(* Logix 5000 project; controller PLC vendor 1 type 14 code 155 rev 30.14; software revision 30.01; part 2 of 4 *)
(* tags used below, declared in another part *)
   Alarm_Word_Compare : DINT[3];
   Alarm_Word_Current : DINT[3];
   Alarm_Word_New : DINT[3];
   Alarm_Word_Previous : DINT[3];
   Bridge_Timer_Gearing_Duration : TIMER;
   Denester : Denester_R2b;
   Depositor : Depositor_R2b;
   IO : IO_R2a;
   MV_Rate : DINT;
   NC_NF : NCNF_R2a;   // NC/NF BITSHIFTS
   OS : INT[10];
   Rates : Rates_R2b;
   Recipe : Recipe_R2c;
   Recipe_Setpoints_DINT : DINT[23,20];
   Recipe_Setpoints_DINT_Temp : DINT[20];
   Recipe_Setpoints_REAL : REAL[23,20];
   Recipe_Setpoints_REAL_Temp : REAL[20];
   Sequencer_Auto : Sequencer_R2a;
   Sequencer_Home : Sequencer_R2a;
   Servo_MC_Bridge_Shift : Axis_MC_R3b;
   System : System_R2e;
(* MainProgram, continued *)

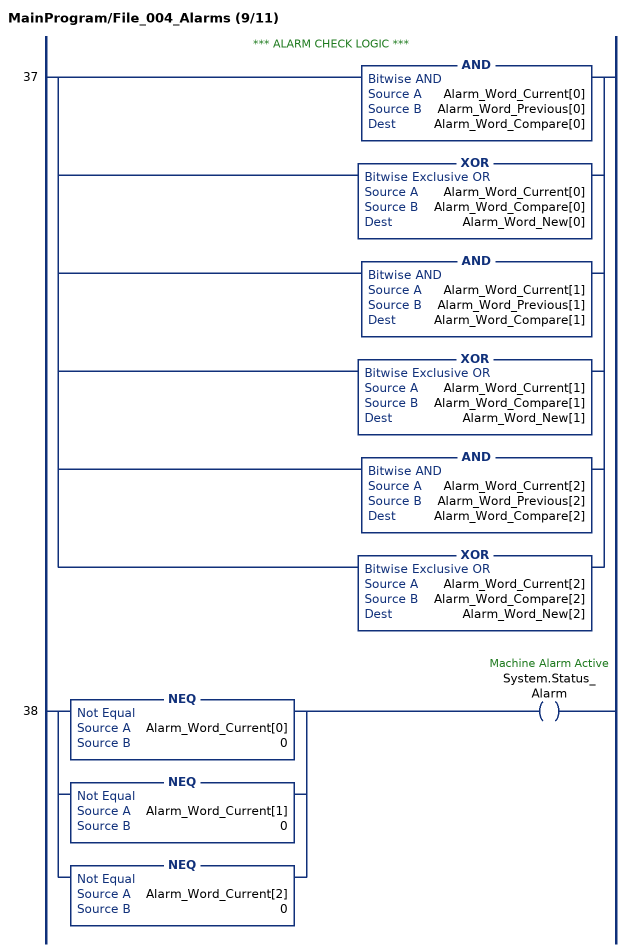
   [picture p24: MainProgram/File_004_Alarms rungs 37-38]
   // *** ALARM CHECK LOGIC ***
   37: [[AND(Alarm_Word_Current[0],Alarm_Word_Previous[0],Alarm_Word_Compare[0]) ,XOR(Alarm_Word_Current[0],Alarm_Word_Compare[0],Alarm_Word_New[0]) ] ,[AND(Alarm_Word_Current[1],Alarm_Word_Previous[1],Alarm_Word_Compare[1]) ,XOR(Alarm_Word_Current[1],Alarm_Word_Compare[1],Alarm_Word_New[1]) ] ,[AND(Alarm_Word_Current[2],Alarm_Word_Previous[2],Alarm_Word_Compare[2]) ,XOR(Alarm_Word_Current[2],Alarm_Word_Compare[2],Alarm_Word_New[2]) ] ];
   38: [NEQ(Alarm_Word_Current[0],0) ,NEQ(Alarm_Word_Current[1],0) ,NEQ(Alarm_Word_Current[2],0) ]OTE(System.Status_Alarm);
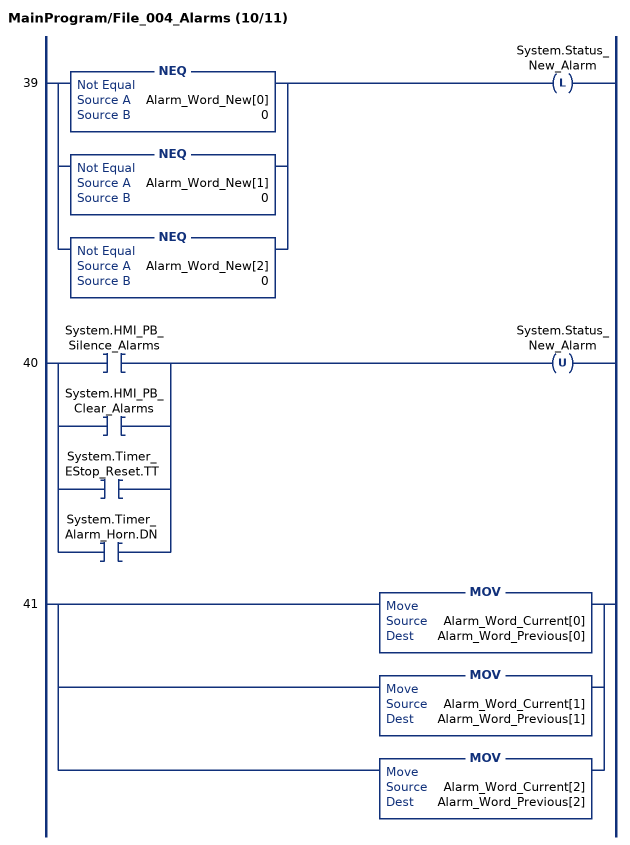
   39: [NEQ(Alarm_Word_New[0],0) ,NEQ(Alarm_Word_New[1],0) ,NEQ(Alarm_Word_New[2],0) ]OTL(System.Status_New_Alarm);
   40: [XIC(System.HMI_PB_Silence_Alarms) ,XIC(System.HMI_PB_Clear_Alarms) ,XIC(System.Timer_EStop_Reset.TT) ,XIC(System.Timer_Alarm_Horn.DN) ]OTU(System.Status_New_Alarm);
   41: [MOV(Alarm_Word_Current[0],Alarm_Word_Previous[0]) ,MOV(Alarm_Word_Current[1],Alarm_Word_Previous[1]) ,MOV(Alarm_Word_Current[2],Alarm_Word_Previous[2]) ];
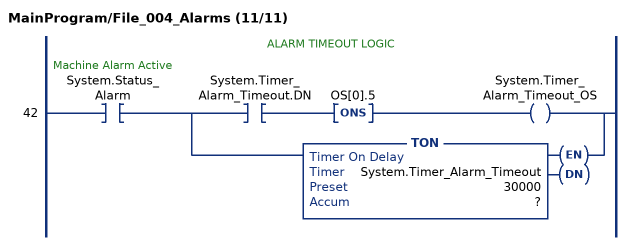
   // ALARM TIMEOUT LOGIC
   42: XIC(System.Status_Alarm)[XIC(System.Timer_Alarm_Timeout.DN) ONS(OS[0].5) OTE(System.Timer_Alarm_Timeout_OS) ,TON(System.Timer_Alarm_Timeout,?,?) ];
END_ROUTINE

ROUTINE File_005_Recipes   (* ladder *)
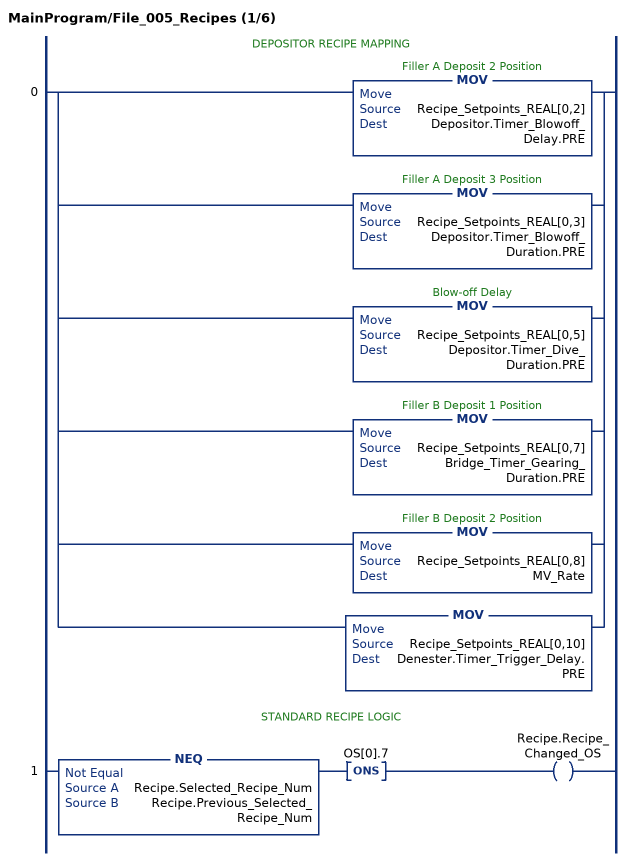
   // DEPOSITOR RECIPE MAPPING
   0: [MOV(Recipe_Setpoints_REAL[0,2],Depositor.Timer_Blowoff_Delay.PRE) ,MOV(Recipe_Setpoints_REAL[0,3],Depositor.Timer_Blowoff_Duration.PRE) ,MOV(Recipe_Setpoints_REAL[0,5],Depositor.Timer_Dive_Duration.PRE) ,MOV(Recipe_Setpoints_REAL[0,7],Bridge_Timer_Gearing_Duration.PRE) ,MOV(Recipe_Setpoints_REAL[0,8],MV_Rate) ,MOV(Recipe_Setpoints_REAL[0,10],Denester.Timer_Trigger_Delay.PRE) ];
   // STANDARD RECIPE LOGIC
   1: NEQ(Recipe.Selected_Recipe_Num,Recipe.Previous_Selected_Recipe_Num)ONS(OS[0].7)OTE(Recipe.Recipe_Changed_OS);
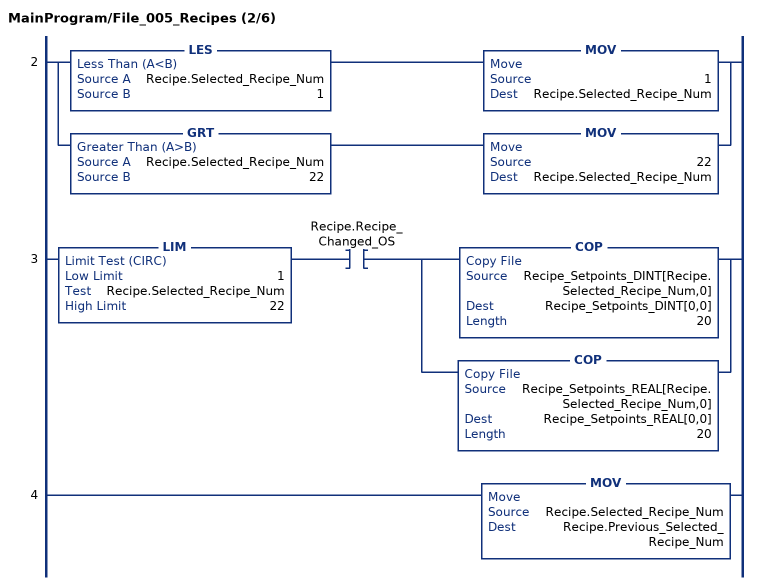
   2: [LES(Recipe.Selected_Recipe_Num,1) MOV(1,Recipe.Selected_Recipe_Num) ,GRT(Recipe.Selected_Recipe_Num,22) MOV(22,Recipe.Selected_Recipe_Num) ];
   3: LIM(1,Recipe.Selected_Recipe_Num,22)XIC(Recipe.Recipe_Changed_OS)[COP(Recipe_Setpoints_DINT[Recipe.Selected_Recipe_Num,0],Recipe_Setpoints_DINT[0,0],20) ,COP(Recipe_Setpoints_REAL[Recipe.Selected_Recipe_Num,0],Recipe_Setpoints_REAL[0,0],20) ];
   4: MOV(Recipe.Selected_Recipe_Num,Recipe.Previous_Selected_Recipe_Num);
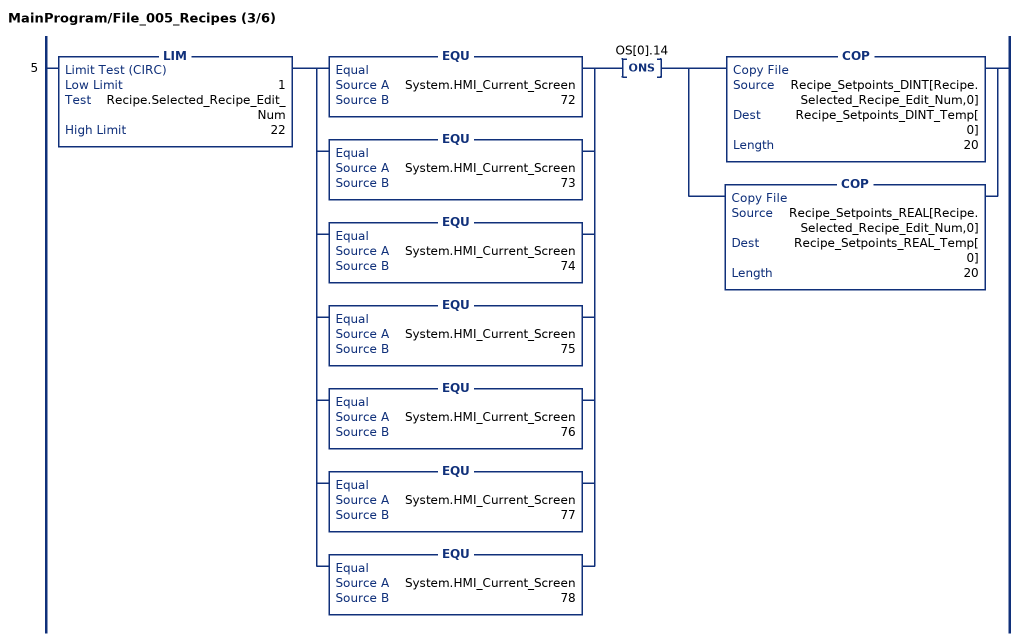
   5: LIM(1,Recipe.Selected_Recipe_Edit_Num,22)[EQU(System.HMI_Current_Screen,72) ,EQU(System.HMI_Current_Screen,73) ,EQU(System.HMI_Current_Screen,74) ,EQU(System.HMI_Current_Screen,75) ,EQU(System.HMI_Current_Screen,76) ,EQU(System.HMI_Current_Screen,77) ,EQU(System.HMI_Current_Screen,78) ]ONS(OS[0].14)[COP(Recipe_Setpoints_DINT[Recipe.Selected_Recipe_Edit_Num,0],Recipe_Setpoints_DINT_Temp[0],20) ,COP(Recipe_Setpoints_REAL[Recipe.Selected_Recipe_Edit_Num,0],Recipe_Setpoints_REAL_Temp[0],20) ];
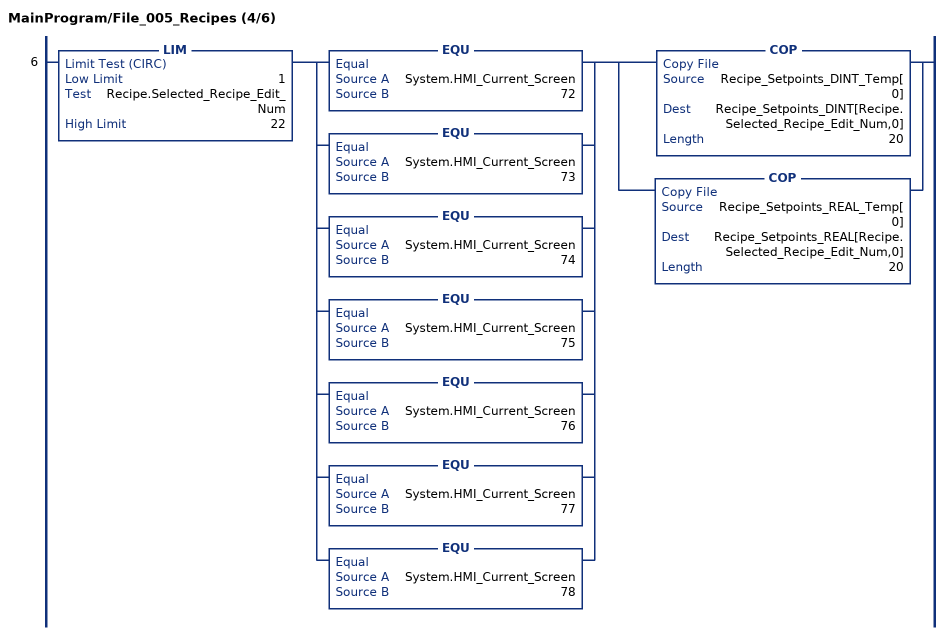
   6: LIM(1,Recipe.Selected_Recipe_Edit_Num,22)[EQU(System.HMI_Current_Screen,72) ,EQU(System.HMI_Current_Screen,73) ,EQU(System.HMI_Current_Screen,74) ,EQU(System.HMI_Current_Screen,75) ,EQU(System.HMI_Current_Screen,76) ,EQU(System.HMI_Current_Screen,77) ,EQU(System.HMI_Current_Screen,78) ][COP(Recipe_Setpoints_DINT_Temp[0],Recipe_Setpoints_DINT[Recipe.Selected_Recipe_Edit_Num,0],20) ,COP(Recipe_Setpoints_REAL_Temp[0],Recipe_Setpoints_REAL[Recipe.Selected_Recipe_Edit_Num,0],20) ];
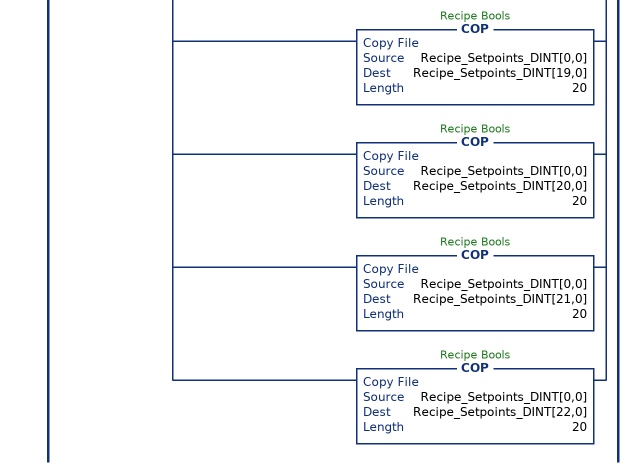
   // RECIPE INITIALIZATION LOGIC
   7: XIC(System.HMI_PB_Recipe_Initialize)[COP(Recipe_Setpoints_DINT[0,0],Recipe_Setpoints_DINT[1,0],20) ,COP(Recipe_Setpoints_DINT[0,0],Recipe_Setpoints_DINT[2,0],20) ,COP(Recipe_Setpoints_DINT[0,0],Recipe_Setpoints_DINT[3,0],20) ,COP(Recipe_Setpoints_DINT[0,0],Recipe_Setpoints_DINT[4,0],20) ,COP(Recipe_Setpoints_DINT[0,0],Recipe_Setpoints_DINT[5,0],20) ,COP(Recipe_Setpoints_DINT[0,0],Recipe_Setpoints_DINT[6,0],20) ,COP(Recipe_Setpoints_DINT[0,0],Recipe_Setpoints_DINT[7,0],20) ,COP(Recipe_Setpoints_DINT[0,0],Recipe_Setpoints_DINT[8,0],20) ,COP(Recipe_Setpoints_DINT[0,0],Recipe_Setpoints_DINT[9,0],20) ,COP(Recipe_Setpoints_DINT[0,0],Recipe_Setpoints_DINT[10,0],20) ,COP(Recipe_Setpoints_DINT[0,0],Recipe_Setpoints_DINT[11,0],20) ,COP(Recipe_Setpoints_DINT[0,0],Recipe_Setpoints_DINT[12,0],20) ,COP(Recipe_Setpoints_DINT[0,0],Recipe_Setpoints_DINT[13,0],20) ,COP(Recipe_Setpoints_DINT[0,0],Recipe_Setpoints_DINT[14,0],20) ,COP(Recipe_Setpoints_DINT[0,0],Recipe_Setpoints_DINT[15,0],20) ,COP(Recipe_Setpoints_DINT[0,0],Recipe_Setpoints_DINT[16,0],20) ,COP(Recipe_Setpoints_DINT[0,0],Recipe_Setpoints_DINT[17,0],20) ,COP(Recipe_Setpoints_DINT[0,0],Recipe_Setpoints_DINT[18,0],20) ,COP(Recipe_Setpoints_DINT[0,0],Recipe_Setpoints_DINT[19,0],20) ,COP(Recipe_Setpoints_DINT[0,0],Recipe_Setpoints_DINT[20,0],20) ,COP(Recipe_Setpoints_DINT[0,0],Recipe_Setpoints_DINT[21,0],20) ,COP(Recipe_Setpoints_DINT[0,0],Recipe_Setpoints_DINT[22,0],20) ];
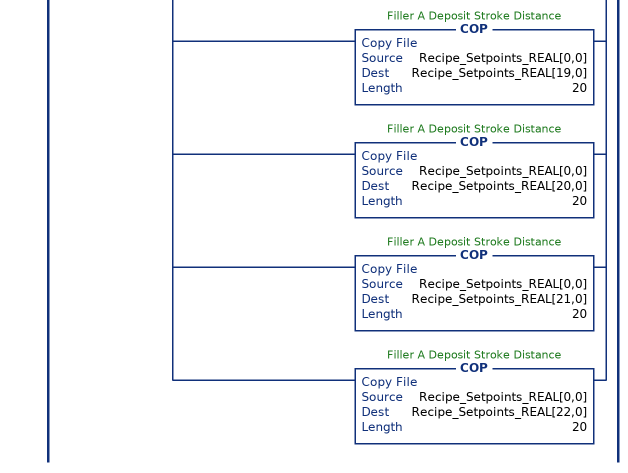
   8: XIC(System.HMI_PB_Recipe_Initialize)[COP(Recipe_Setpoints_REAL[0,0],Recipe_Setpoints_REAL[1,0],20) ,COP(Recipe_Setpoints_REAL[0,0],Recipe_Setpoints_REAL[2,0],20) ,COP(Recipe_Setpoints_REAL[0,0],Recipe_Setpoints_REAL[3,0],20) ,COP(Recipe_Setpoints_REAL[0,0],Recipe_Setpoints_REAL[4,0],20) ,COP(Recipe_Setpoints_REAL[0,0],Recipe_Setpoints_REAL[5,0],20) ,COP(Recipe_Setpoints_REAL[0,0],Recipe_Setpoints_REAL[6,0],20) ,COP(Recipe_Setpoints_REAL[0,0],Recipe_Setpoints_REAL[7,0],20) ,COP(Recipe_Setpoints_REAL[0,0],Recipe_Setpoints_REAL[8,0],20) ,COP(Recipe_Setpoints_REAL[0,0],Recipe_Setpoints_REAL[9,0],20) ,COP(Recipe_Setpoints_REAL[0,0],Recipe_Setpoints_REAL[10,0],20) ,COP(Recipe_Setpoints_REAL[0,0],Recipe_Setpoints_REAL[11,0],20) ,COP(Recipe_Setpoints_REAL[0,0],Recipe_Setpoints_REAL[12,0],20) ,COP(Recipe_Setpoints_REAL[0,0],Recipe_Setpoints_REAL[13,0],20) ,COP(Recipe_Setpoints_REAL[0,0],Recipe_Setpoints_REAL[14,0],20) ,COP(Recipe_Setpoints_REAL[0,0],Recipe_Setpoints_REAL[15,0],20) ,COP(Recipe_Setpoints_REAL[0,0],Recipe_Setpoints_REAL[16,0],20) ,COP(Recipe_Setpoints_REAL[0,0],Recipe_Setpoints_REAL[17,0],20) ,COP(Recipe_Setpoints_REAL[0,0],Recipe_Setpoints_REAL[18,0],20) ,COP(Recipe_Setpoints_REAL[0,0],Recipe_Setpoints_REAL[19,0],20) ,COP(Recipe_Setpoints_REAL[0,0],Recipe_Setpoints_REAL[20,0],20) ,COP(Recipe_Setpoints_REAL[0,0],Recipe_Setpoints_REAL[21,0],20) ,COP(Recipe_Setpoints_REAL[0,0],Recipe_Setpoints_REAL[22,0],20) ];
END_ROUTINE

ROUTINE File_006_Status   (* ladder *)
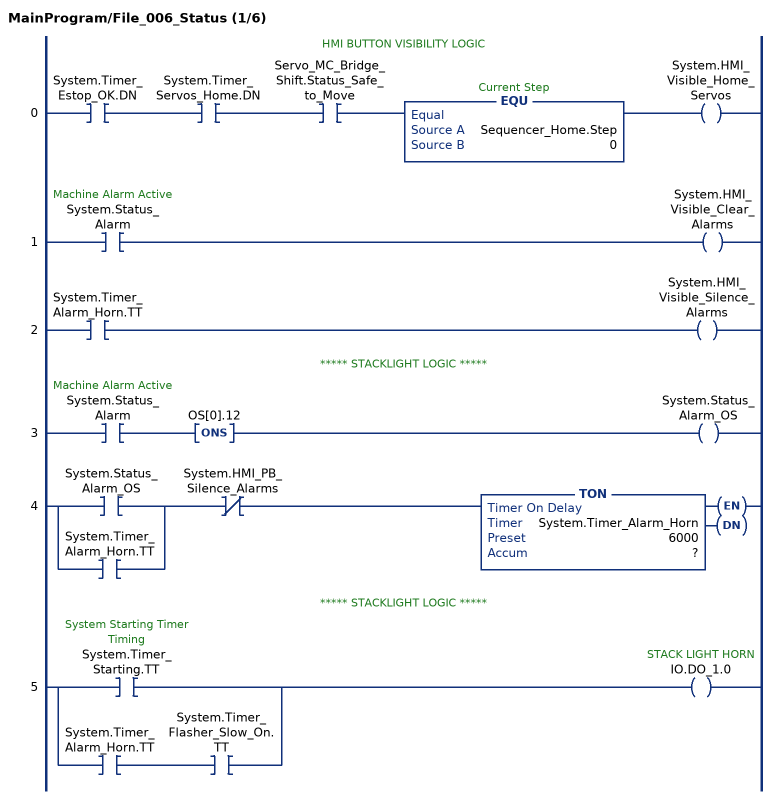
   // HMI BUTTON VISIBILITY LOGIC
   0: XIC(System.Timer_Estop_OK.DN)XIC(System.Timer_Servos_Home.DN)XIC(Servo_MC_Bridge_Shift.Status_Safe_to_Move)EQU(Sequencer_Home.Step,0)OTE(System.HMI_Visible_Home_Servos);
   1: XIC(System.Status_Alarm)OTE(System.HMI_Visible_Clear_Alarms);
   2: XIC(System.Timer_Alarm_Horn.TT)OTE(System.HMI_Visible_Silence_Alarms);
   // ***** STACKLIGHT LOGIC *****
   3: XIC(System.Status_Alarm)ONS(OS[0].12)OTE(System.Status_Alarm_OS);
   4: [XIC(System.Status_Alarm_OS) ,XIC(System.Timer_Alarm_Horn.TT) ]XIO(System.HMI_PB_Silence_Alarms)TON(System.Timer_Alarm_Horn,?,?);
   // ***** STACKLIGHT LOGIC *****
   5: [XIC(System.Timer_Starting.TT) ,XIC(System.Timer_Alarm_Horn.TT) XIC(System.Timer_Flasher_Slow_On.TT) ]OTE(IO.DO_1.0);
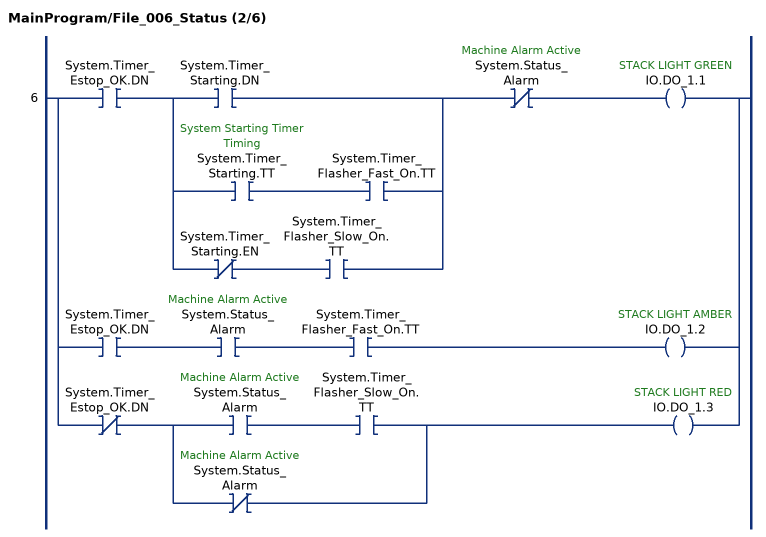
   6: [XIC(System.Timer_Estop_OK.DN) [XIC(System.Timer_Starting.DN) ,XIC(System.Timer_Starting.TT) XIC(System.Timer_Flasher_Fast_On.TT) ,XIO(System.Timer_Starting.EN) XIC(System.Timer_Flasher_Slow_On.TT) ] XIO(System.Status_Alarm) OTE(IO.DO_1.1) ,XIC(System.Timer_Estop_OK.DN) XIC(System.Status_Alarm) XIC(System.Timer_Flasher_Fast_On.TT) OTE(IO.DO_1.2) ,XIO(System.Timer_Estop_OK.DN) [XIC(System.Status_Alarm) XIC(System.Timer_Flasher_Slow_On.TT) ,XIO(System.Status_Alarm) ] OTE(IO.DO_1.3) ];
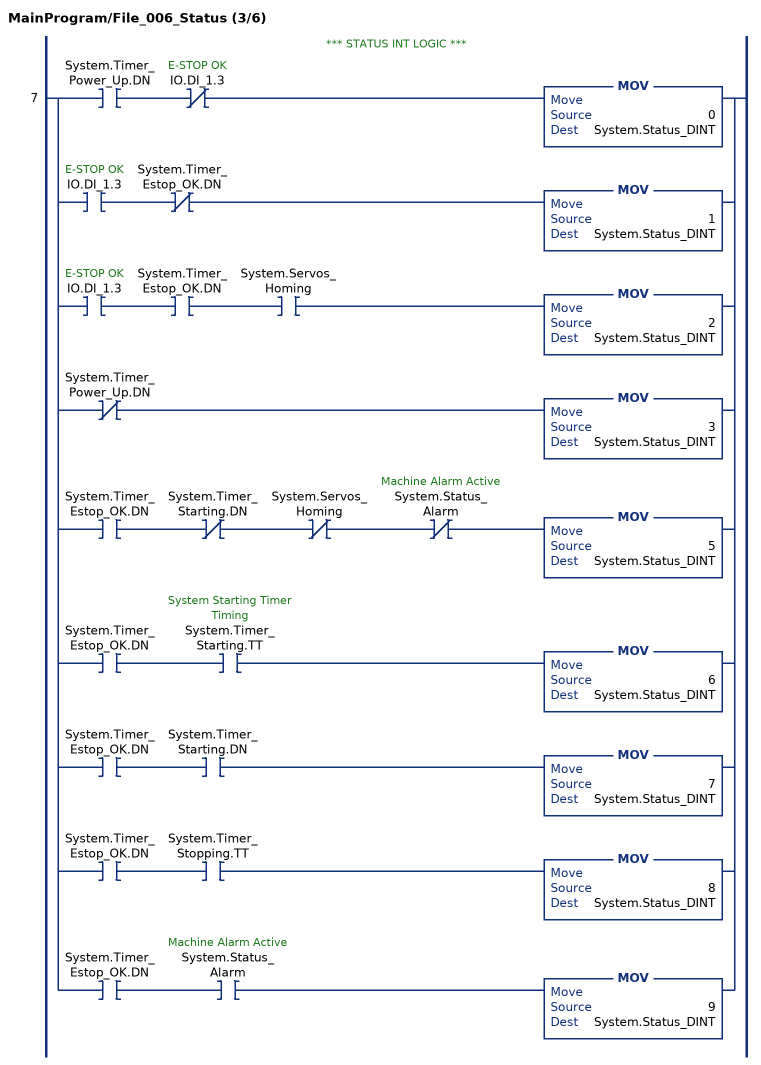
   // *** STATUS INT LOGIC ***
   7: [XIC(System.Timer_Power_Up.DN) XIO(IO.DI_1.3) MOV(0,System.Status_DINT) ,XIC(IO.DI_1.3) XIO(System.Timer_Estop_OK.DN) MOV(1,System.Status_DINT) ,XIC(IO.DI_1.3) XIC(System.Timer_Estop_OK.DN) XIC(System.Servos_Homing) MOV(2,System.Status_DINT) ,XIO(System.Timer_Power_Up.DN) MOV(3,System.Status_DINT) ,XIC(System.Timer_Estop_OK.DN) XIO(System.Timer_Starting.DN) XIO(System.Servos_Homing) XIO(System.Status_Alarm) MOV(5,System.Status_DINT) ,XIC(System.Timer_Estop_OK.DN) XIC(System.Timer_Starting.TT) MOV(6,System.Status_DINT) ,XIC(System.Timer_Estop_OK.DN) XIC(System.Timer_Starting.DN) MOV(7,System.Status_DINT) ,XIC(System.Timer_Estop_OK.DN) XIC(System.Timer_Stopping.TT) MOV(8,System.Status_DINT) ,XIC(System.Timer_Estop_OK.DN) XIC(System.Status_Alarm) MOV(9,System.Status_DINT) ];
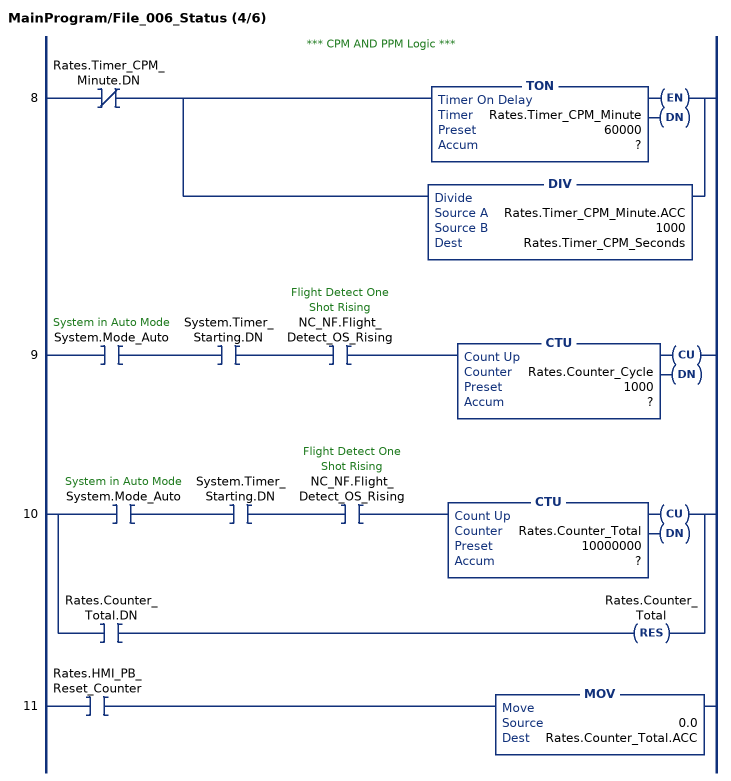
   // *** CPM AND PPM Logic ***
   8: XIO(Rates.Timer_CPM_Minute.DN)[TON(Rates.Timer_CPM_Minute,?,?) ,DIV(Rates.Timer_CPM_Minute.ACC,1000,Rates.Timer_CPM_Seconds) ];
   9: XIC(System.Mode_Auto)XIC(System.Timer_Starting.DN)XIC(NC_NF.Flight_Detect_OS_Rising)CTU(Rates.Counter_Cycle,?,?);
   10: [XIC(System.Mode_Auto) XIC(System.Timer_Starting.DN) XIC(NC_NF.Flight_Detect_OS_Rising) CTU(Rates.Counter_Total,?,?) ,XIC(Rates.Counter_Total.DN) RES(Rates.Counter_Total) ];
   11: XIC(Rates.HMI_PB_Reset_Counter)MOV(0.0,Rates.Counter_Total.ACC);
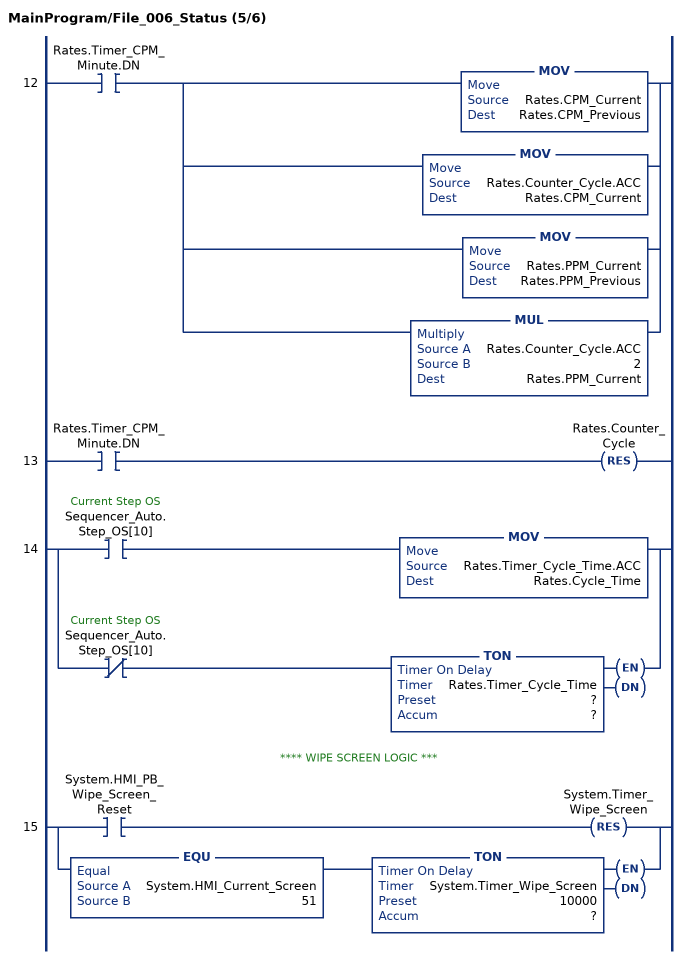
   12: XIC(Rates.Timer_CPM_Minute.DN)[MOV(Rates.CPM_Current,Rates.CPM_Previous) ,MOV(Rates.Counter_Cycle.ACC,Rates.CPM_Current) ,MOV(Rates.PPM_Current,Rates.PPM_Previous) ,MUL(Rates.Counter_Cycle.ACC,2,Rates.PPM_Current) ];
   13: XIC(Rates.Timer_CPM_Minute.DN)RES(Rates.Counter_Cycle);
   14: [XIC(Sequencer_Auto.Step_OS[10]) MOV(Rates.Timer_Cycle_Time.ACC,Rates.Cycle_Time) ,XIO(Sequencer_Auto.Step_OS[10]) TON(Rates.Timer_Cycle_Time,?,?) ];
   // **** WIPE SCREEN LOGIC ***
   15: [XIC(System.HMI_PB_Wipe_Screen_Reset) RES(System.Timer_Wipe_Screen) ,EQU(System.HMI_Current_Screen,51) TON(System.Timer_Wipe_Screen,?,?) ];
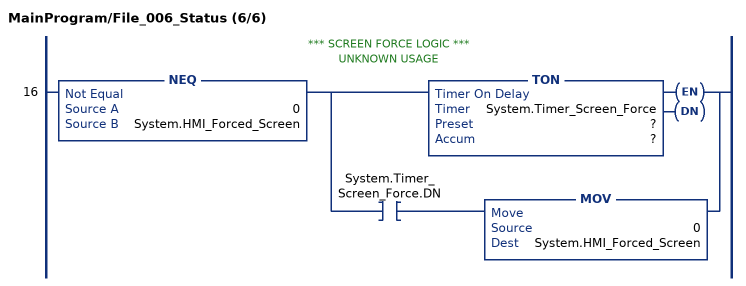
   // *** SCREEN FORCE LOGIC ***
   // UNKNOWN USAGE
   16: NEQ(0,System.HMI_Forced_Screen)[TON(System.Timer_Screen_Force,?,?) ,XIC(System.Timer_Screen_Force.DN) MOV(0,System.HMI_Forced_Screen) ];
END_ROUTINE

ROUTINE File_007_NC_NF   (* ladder *)
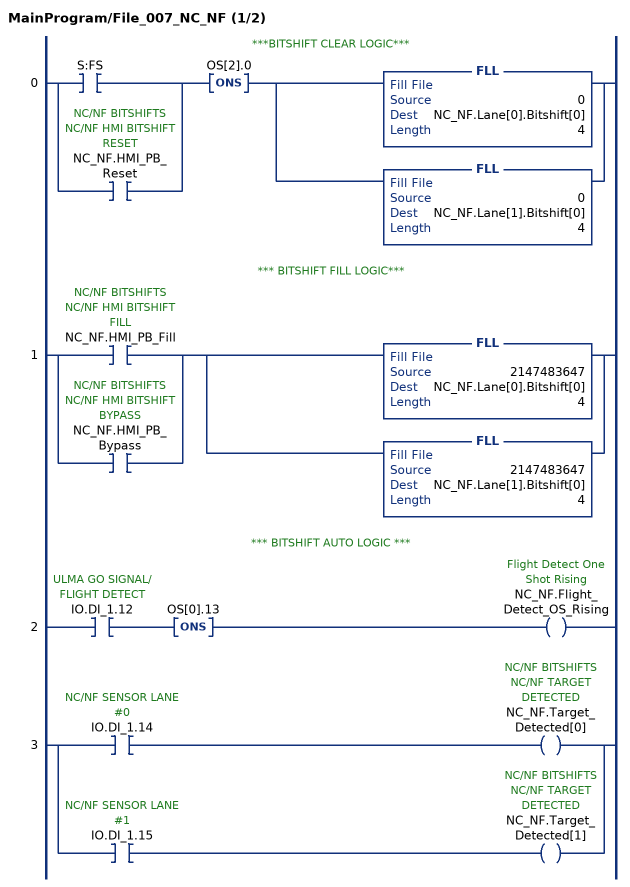
   // ***BITSHIFT CLEAR LOGIC***
   0: [XIC(S:FS) ,XIC(NC_NF.HMI_PB_Reset) ]ONS(OS[2].0)[FLL(0,NC_NF.Lane[0].Bitshift[0],4) ,FLL(0,NC_NF.Lane[1].Bitshift[0],4) ];
   // *** BITSHIFT FILL LOGIC***
   1: [XIC(NC_NF.HMI_PB_Fill) ,XIC(NC_NF.HMI_PB_Bypass) ][FLL(2147483647,NC_NF.Lane[0].Bitshift[0],4) ,FLL(2147483647,NC_NF.Lane[1].Bitshift[0],4) ];
   // *** BITSHIFT AUTO LOGIC ***
   2: XIC(IO.DI_1.12)ONS(OS[0].13)OTE(NC_NF.Flight_Detect_OS_Rising);
   3: [XIC(IO.DI_1.14) OTE(NC_NF.Target_Detected[0]) ,XIC(IO.DI_1.15) OTE(NC_NF.Target_Detected[1]) ];
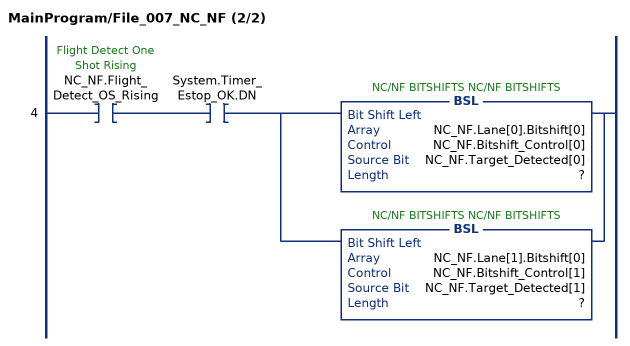
   4: XIC(NC_NF.Flight_Detect_OS_Rising)XIC(System.Timer_Estop_OK.DN)[BSL(NC_NF.Lane[0].Bitshift[0],NC_NF.Bitshift_Control[0],NC_NF.Target_Detected[0],?) ,BSL(NC_NF.Lane[1].Bitshift[0],NC_NF.Bitshift_Control[1],NC_NF.Target_Detected[1],?) ];
END_ROUTINE

ROUTINE File_010_Digital_Inputs   (* ladder *)
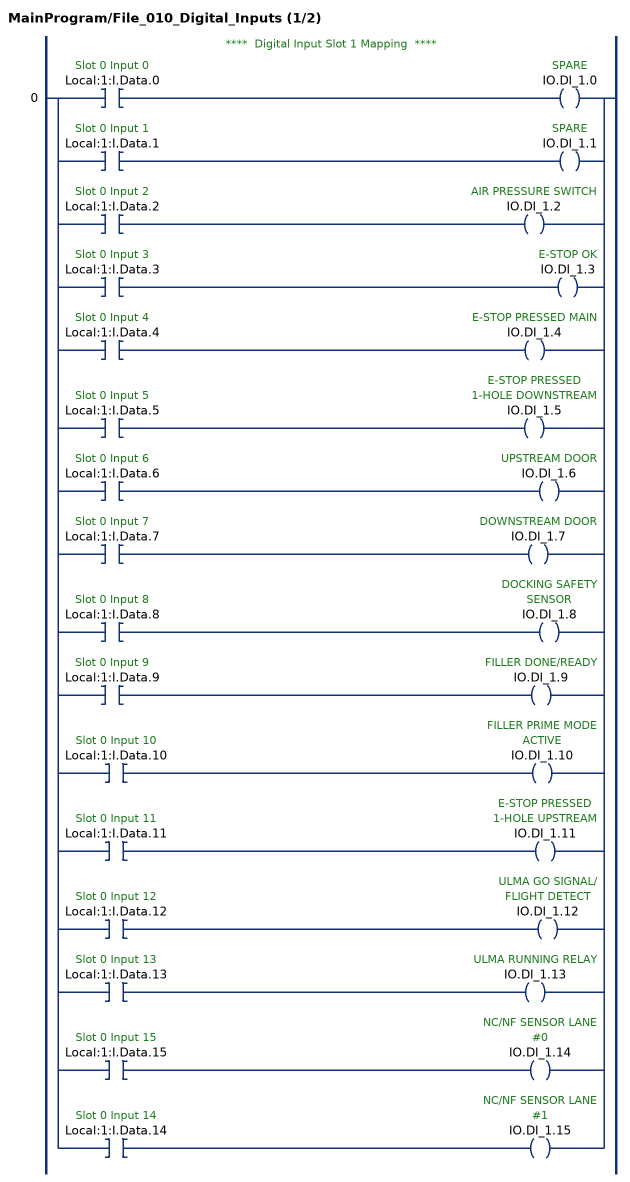
   // ****  Digital Input Slot 1 Mapping  ****
   0: [XIC(Local:1:I.Data.0) OTE(IO.DI_1.0) ,XIC(Local:1:I.Data.1) OTE(IO.DI_1.1) ,XIC(Local:1:I.Data.2) OTE(IO.DI_1.2) ,XIC(Local:1:I.Data.3) OTE(IO.DI_1.3) ,XIC(Local:1:I.Data.4) OTE(IO.DI_1.4) ,XIC(Local:1:I.Data.5) OTE(IO.DI_1.5) ,XIC(Local:1:I.Data.6) OTE(IO.DI_1.6) ,XIC(Local:1:I.Data.7) OTE(IO.DI_1.7) ,XIC(Local:1:I.Data.8) OTE(IO.DI_1.8) ,XIC(Local:1:I.Data.9) OTE(IO.DI_1.9) ,XIC(Local:1:I.Data.10) OTE(IO.DI_1.10) ,XIC(Local:1:I.Data.11) OTE(IO.DI_1.11) ,XIC(Local:1:I.Data.12) OTE(IO.DI_1.12) ,XIC(Local:1:I.Data.13) OTE(IO.DI_1.13) ,XIC(Local:1:I.Data.15) OTE(IO.DI_1.14) ,XIC(Local:1:I.Data.14) OTE(IO.DI_1.15) ];
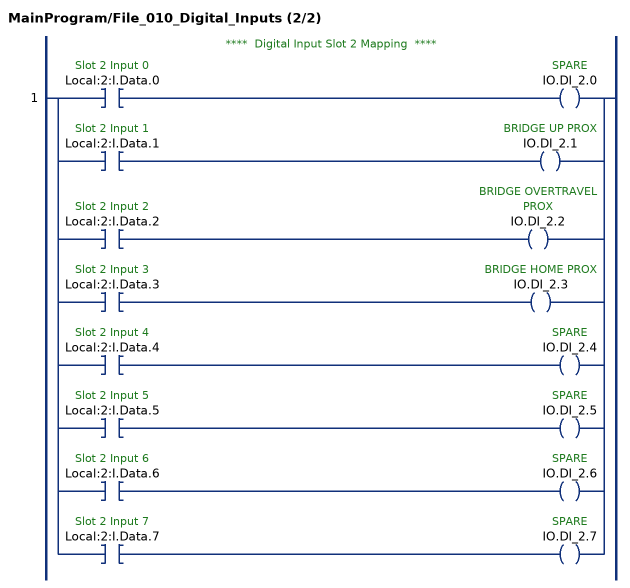
   // ****  Digital Input Slot 2 Mapping  ****
   1: [XIC(Local:2:I.Data.0) OTE(IO.DI_2.0) ,XIC(Local:2:I.Data.1) OTE(IO.DI_2.1) ,XIC(Local:2:I.Data.2) OTE(IO.DI_2.2) ,XIC(Local:2:I.Data.3) OTE(IO.DI_2.3) ,XIC(Local:2:I.Data.4) OTE(IO.DI_2.4) ,XIC(Local:2:I.Data.5) OTE(IO.DI_2.5) ,XIC(Local:2:I.Data.6) OTE(IO.DI_2.6) ,XIC(Local:2:I.Data.7) OTE(IO.DI_2.7) ];
END_ROUTINE
